// ---- POUs/Machine/CleaningStation/_VISU_CleanPU.TcVIS
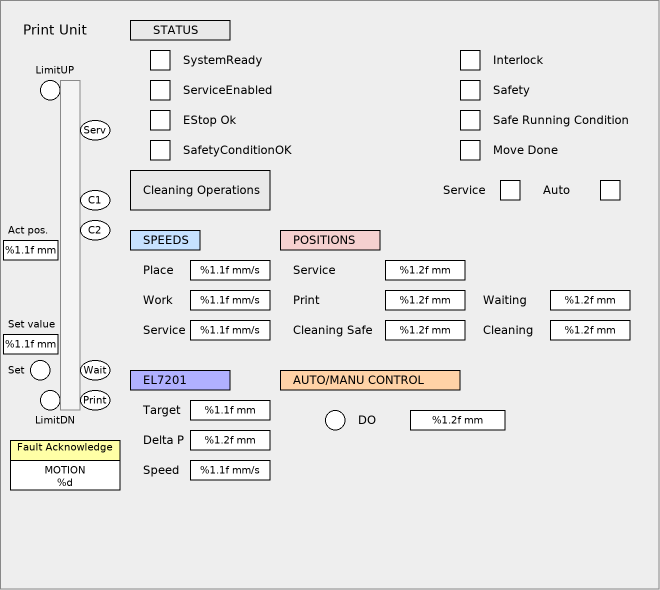
VISUALIZATION _VISU_CleanPU  // 660x590
VAR_IN_OUT
  mInst  : FB_CleaningMotorAxisPU;
END_VAR
    Rectangle (0,0 660x590)
    Polyline (200,380)
    Polyline (130,240)
    Rectangle (130,170 140x40)
    Rectangle (130,370 100x20)
    Rectangle (280,370 180x20)
    Rectangle (280,230 100x20)
    Rectangle (130,230 70x20)
    Rectangle (130,20 100x20)
    Rectangle (20,20 100x20), "Print Unit"
    Polyline (130,30)
    Polyline (230,30)
    Rectangle (150,20 60x20), "STATUS"
    RoundedRectangle (150,80 20x20), colour toggle: mInst.bI_UsrService
    RoundedRectangle (150,110 20x20), colour toggle: NOT mInst.bI_Emergency
    RoundedRectangle (150,140 20x20), colour toggle: mInst.bI_SafetyOk
    RoundedRectangle (460,140 20x20), colour toggle: NOT mInst.bL_Busy
    RoundedRectangle (150,50 20x20), colour toggle: mInst.bI_MachineReady
    Rectangle (180,50 120x20), "SystemReady"
    Rectangle (180,80 120x20), "ServiceEnabled"
    Rectangle (180,110 120x20), "EStop Ok"
    Rectangle (180,140 120x20), "SafetyConditionOK"
    Rectangle (490,140 90x20), "Move Done"
    Rectangle (290,370 170x20), "AUTO/MANU CONTROL"
    Polyline (450,380)
    Rectangle (30,60 50x20), "LimitUP"
    Ellipse (40,80 20x20), colour toggle: NOT mInst.bI_SensorTop
    Ellipse (40,390 20x20), colour toggle: NOT mInst.bI_SensorBottom
    Rectangle (30,410 50x20), "LimitDN"
    Scrollbar (60,80 20x330)
        p2245068023: 0.5
        p1057716461: mInst.fB_Axis.fO_ActualPosition
    Rectangle (140,230 70x20), "SPEEDS"
    Rectangle (190,260 80x20), "%1.1f mm/s", text variable: mInst.sI_SpeedDef.fP_PlaceSpeed
        OnMouseDown: write the text variable via VisuDialogs.Numpad
    Rectangle (190,290 80x20), "%1.1f mm/s", text variable: mInst.sI_SpeedDef.fP_WorkSpeed
        OnMouseDown: write the text variable via VisuDialogs.Numpad
    Rectangle (190,320 80x20), "%1.1f mm/s", text variable: mInst.sI_SpeedDef.fP_ServiceSpeed
        OnMouseDown: write the text variable via VisuDialogs.Numpad
    Rectangle (140,260 45x20), "Place"
    Rectangle (140,290 45x20), "Work"
    Rectangle (140,320 45x20), "Service"
        OnMouseDown: write the text variable via Edit
    Rectangle (290,260 90x20), "Service"
    Rectangle (290,290 90x20), "Print"
    Polyline (350,240)
    Rectangle (290,230 90x20), "POSITIONS"
    Rectangle (190,400 80x20), "%1.1f mm", text variable: 1000 * mInst.fB_Axis.fI_TargetPosition
    RoundedRectangle (460,80 20x20), colour toggle: mInst.bI_SafeToMove
    Rectangle (490,80 120x20), "Safety"
    RoundedRectangle (460,50 20x20), colour toggle: mInst.bI_SafeToMove
    Rectangle (490,50 120x20), "Interlock"
    Rectangle (5,360 25x20), "Set"
    Ellipse (30,360 20x20), colour toggle: mInst.fB_Axis.bI_SetPosition
        toggle mInst.fB_Axis.bI_SetPosition
    Rectangle (3,240 55x20), "%1.1f mm", text variable: 1000 * mInst.fB_Axis.fO_ActualPosition
    Rectangle (290,320 90x20), "Cleaning Safe"
    Rectangle (385,320 80x20), "%1.2f mm", text variable: mInst.fI_PositionClean1
        OnMouseDown: write the text variable via VisuDialogs.Numpad
    Rectangle (140,400 45x20), "Target"
    Rectangle (140,460 45x20), "Speed"
    Rectangle (190,460 80x20), "%1.1f mm/s", text variable: 1000 * mInst.fB_Axis.fI_SpeedLimit
    Rectangle (140,370 90x20), "EL7201"
    Rectangle (140,430 45x20), "Delta P"
    Rectangle (190,430 80x20), "%1.2f mm", text variable: 1000 * mInst.fB_Axis.fL_Delta_P
    Ellipse (80,120 30x20), "Serv", colour toggle: mInst.pInPosService
    Ellipse (80,220 30x20), "C2", colour toggle: mInst.pInPosClean2
    Ellipse (80,190 30x20), "C1", colour toggle: mInst.pInPosClean1
    Ellipse (80,360 30x20), "Wait", colour toggle: mInst.pInPosWait
    Ellipse (80,390 30x20), "Print", colour toggle: mInst.pInPosPrint
    Polyline (640,160)
    Rectangle (140,180 140x20), "Cleaning Operations"
    Polyline (270,200)
    RoundedRectangle (460,110 20x20), colour toggle: mInst.bL_SafeRunningCondition
    Rectangle (490,110 140x20), "Safe Running Condition"
    RoundedRectangle (600,180 20x20), colour toggle: mInst.bI_UsrAutoMode
    Rectangle (540,180 55x20), "Auto"
    Polyline (340,80)
    Rectangle (10,440 110x50), "Fault Acknowledge", colour toggle: (mInst.wL_ErrorCode) <> 0
    RoundedRectangle (10,460 110x30), "%d", text variable: mInst.wL_ErrorCode
        tap mInst.sADS_CleanAxis.bI_FaultAck
    RoundedRectangle (10,460 110x20), "MOTION"
    Rectangle (3,334 55x20), "%1.1f mm", text variable: mInst.fL_SetPositionValue
        OnMouseDown: write the text variable via VisuDialogs.Numpad
    Rectangle (480,320 65x20), "Cleaning"
    Rectangle (550,320 80x20), "%1.2f mm", text variable: mInst.fI_PositionClean2
        OnMouseDown: write the text variable via VisuDialogs.Numpad
    RoundedRectangle (500,180 20x20), colour toggle: mInst.bI_UsrService
    Rectangle (440,180 55x20), "Service"
    Rectangle (410,410 95x20), "%1.2f mm", text variable: mInst.sADS_CleanAxis.fI_ManualTargetPos
        OnMouseDown: write the text variable via VisuDialogs.Numpad, min mInst.sADS_CleanAxis.sO_AxisPosition.fC_Min, max mInst.sADS_CleanAxis.sO_AxisPosition.fC_Max
    Rectangle (355,410 50x20), "DO"
    Ellipse (325,410 20x20), colour toggle: mInst.sADS_CleanAxis.bI_ManualMove, input disabled if: NOT mInst.sADS_CleanAxis.bO_ManualMoveCanEx
        toggle mInst.sADS_CleanAxis.bI_ManualMove
    Rectangle (385,260 80x20), "%1.2f mm", text variable: mInst.fI_PositionService
        OnMouseDown: write the text variable via VisuDialogs.Numpad
    Rectangle (385,290 80x20), "%1.2f mm", text variable: mInst.fL_PrintPositionMM
        OnMouseDown: write the text variable via VisuDialogs.Numpad, min 0.8, max 2.5
    Rectangle (480,290 65x20), "Waiting"
    Rectangle (550,290 80x20), "%1.2f mm", text variable: mInst.fI_PositionWait
        OnMouseDown: write the text variable via VisuDialogs.Numpad
    Rectangle (5,314 50x20), "Set value"
    Rectangle (5,220 50x20), "Act pos."
END_VISUALIZATION

// ---- POUs/Machine/CleaningStation/_VISU_CleanSequence.TcVIS
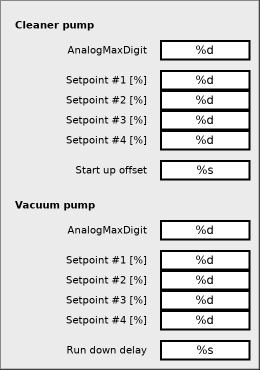
VISUALIZATION _VISU_CleanSequence  // 260x370
    Rectangle (0,0 260x370)
    Rectangle (160,40 90x20), "%d", text variable: PRG_MACHINE.fb_CleaningControl[PRG_MACHINE.iL_Sel_Module].fb_CleaningValvePump.lR_AnalogMaxDigitCleanerPump
        OnMouseDown: write the text variable via Default
    Rectangle (10,40 140x20), "AnalogMaxDigit"
    Rectangle (12,15 131x20), "Cleaner pump"
    Rectangle (160,70 90x20), "%d", text variable: PRG_MACHINE.fb_CleaningControl[PRG_MACHINE.iL_Sel_Module].fb_CleaningValvePump.lR_SetPoint1CleanerPump
        OnMouseDown: write the text variable via Default, min 0, max 100
    Rectangle (10,70 140x20), "Setpoint #1 [%]"
    Rectangle (160,90 90x20), "%d", text variable: PRG_MACHINE.fb_CleaningControl[PRG_MACHINE.iL_Sel_Module].fb_CleaningValvePump.lR_SetPoint2CleanerPump
        OnMouseDown: write the text variable via Default, min 0, max 100
    Rectangle (10,90 140x20), "Setpoint #2 [%]"
    Rectangle (160,110 90x20), "%d", text variable: PRG_MACHINE.fb_CleaningControl[PRG_MACHINE.iL_Sel_Module].fb_CleaningValvePump.lR_SetPoint3CleanerPump
        OnMouseDown: write the text variable via Default, min 0, max 100
    Rectangle (10,110 140x20), "Setpoint #3 [%]"
    Rectangle (160,130 90x20), "%d", text variable: PRG_MACHINE.fb_CleaningControl[PRG_MACHINE.iL_Sel_Module].fb_CleaningValvePump.lR_SetPoint4CleanerPump
        OnMouseDown: write the text variable via Default, min 0, max 100
    Rectangle (10,130 140x20), "Setpoint #4 [%]"
    Rectangle (160,220 90x20), "%d", text variable: PRG_MACHINE.fb_CleaningControl[PRG_MACHINE.iL_Sel_Module].fb_CleaningValvePump.lR_AnalogMaxDigitVacuumPump
        OnMouseDown: write the text variable via Default
    Rectangle (10,220 140x20), "AnalogMaxDigit"
    Rectangle (12,195 131x20), "Vacuum pump"
    Rectangle (160,250 90x20), "%d", text variable: PRG_MACHINE.fb_CleaningControl[PRG_MACHINE.iL_Sel_Module].fb_CleaningValvePump.lR_SetPoint1VacuumPump
        OnMouseDown: write the text variable via Default, min 0, max 100
    Rectangle (10,250 140x20), "Setpoint #1 [%]"
    Rectangle (160,270 90x20), "%d", text variable: PRG_MACHINE.fb_CleaningControl[PRG_MACHINE.iL_Sel_Module].fb_CleaningValvePump.lR_SetPoint2VacuumPump
        OnMouseDown: write the text variable via Default, min 0, max 100
    Rectangle (10,270 140x20), "Setpoint #2 [%]"
    Rectangle (160,290 90x20), "%d", text variable: PRG_MACHINE.fb_CleaningControl[PRG_MACHINE.iL_Sel_Module].fb_CleaningValvePump.lR_SetPoint3VacuumPump
        OnMouseDown: write the text variable via Default, min 0, max 100
    Rectangle (10,290 140x20), "Setpoint #3 [%]"
    Rectangle (160,310 90x20), "%d", text variable: PRG_MACHINE.fb_CleaningControl[PRG_MACHINE.iL_Sel_Module].fb_CleaningValvePump.lR_SetPoint4VacuumPump
        OnMouseDown: write the text variable via Default, min 0, max 100
    Rectangle (10,310 140x20), "Setpoint #4 [%]"
    Rectangle (160,160 90x20), "%s", text variable: PRG_MACHINE.fb_CleaningControl[PRG_MACHINE.iL_Sel_Module].fb_CleaningValvePump.tR_CleanerPumpOffset
        OnMouseDown: write the text variable via Default
    Rectangle (10,160 140x20), "Start up offset"
    Rectangle (160,340 90x20), "%s", text variable: PRG_MACHINE.fb_CleaningControl[PRG_MACHINE.iL_Sel_Module].fb_CleaningValvePump.tR_VacuumPumpDelay
        OnMouseDown: write the text variable via Default
    Rectangle (10,340 140x20), "Run down delay"
END_VISUALIZATION

// ---- POUs/Machine/EffectiveEncoderResolutionDetection/_VISU_EffectiveEncoderResolutionDetection.TcVIS
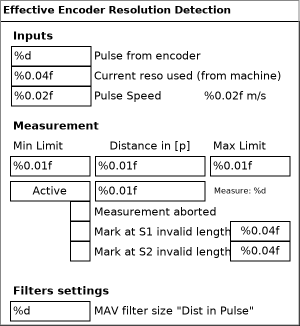
VISUALIZATION _VISU_EffectiveEncoderResolutionDetection  // 300x326
VAR_IN_OUT
	mInst : FB_EffectiveEncoderResolutionDetection;
END_VAR
    Rectangle (0,21 300x305)
    Rectangle (10,116 100x20), "Measurement"
    RoundedRectangle (10,181 80x20), "Active", colour toggle: mInst.bMeasurementActive
    Rectangle (95,156 110x20), "%0.01f", text variable: mInst.fDisInPulse
    Rectangle (95,136 110x20), "Distance in [p]"
    Rectangle (91,86 200x20), "Pulse Speed"
    Rectangle (11,86 80x20), "%0.02f", text variable: mInst.fSpeedPulse
    Rectangle (91,46 200x20), "Pulse from encoder"
    Rectangle (11,46 80x20), "%d", text variable: mInst.nPulse
    Rectangle (11,66 80x20), "%0.04f", text variable: mInst.fCurrentResolution, input disabled if: TRUE
    Rectangle (91,66 200x20), "Current reso used (from machine)"
    Rectangle (10,281 100x20), "Filters settings"
    Rectangle (91,301 200x20), "MAV filter size "Dist in Pulse""
    Rectangle (10,301 80x20), "%d", text variable: mInst.nDisInPulseFilterSz, input disabled if: TRUE
    Rectangle (10,26 100x20), "Inputs"
    Rectangle (0,0 240x20), "Effective Encoder Resolution Detection"
    Rectangle (211,181 80x20), "Measure: %d", tooltip "measurement counter", text variable: mInst.nMeasurementCounter
    Rectangle (10,156 80x20), "%0.01f", tooltip "Limits from machine", text variable: mInst.fEncoderPulseDistMin, colour toggle: mInst.bLower, input disabled if: TRUE
    Rectangle (210,156 80x20), "%0.01f", tooltip "Limits from machine", text variable: mInst.fEncoderPulseDistMax, colour toggle: mInst.bHigher, input disabled if: TRUE
    Rectangle (10,136 80x20), "Min Limit"
    Rectangle (210,136 80x20), "Max Limit"
    RoundedRectangle (70,201 20x20), colour toggle: mInst.bAborted
    Rectangle (91,202 200x20), "Measurement aborted"
    RoundedRectangle (70,221 20x20), colour toggle: mInst.bMarkInvalidLength_S1
    Rectangle (91,222 200x20), "Mark at S1 invalid length"
    RoundedRectangle (70,241 20x20), colour toggle: mInst.bMarkInvalidLength_S2
    Rectangle (91,242 200x20), "Mark at S2 invalid length"
    Rectangle (230,221 60x20), "%0.04f", tooltip "Mark length in [mm], minimum length=%0.02f [mm]", text variable: mInst.nMarkLength_S1/1000, colour toggle: mInst.bMarkInvalidLength_S1
        p4168582468: mInst.nC_MinMarkLength/1000
    Rectangle (230,241 60x20), "%0.04f", tooltip "Mark length in [mm], minimum length=%0.02f [mm]", text variable: mInst.nMarkLength_S2/1000, colour toggle: mInst.bMarkInvalidLength_S2
        p4168582468: mInst.nC_MinMarkLength/1000
    Rectangle (95,181 110x20), "%0.01f", text variable: mInst.nCurrentDistActive
    Rectangle (201,86 80x20), "%0.02f m/s", text variable: mInst.fSpeedUm_s/1_000_000, input disabled if: TRUE
END_VISUALIZATION

// ---- POUs/Machine/ExhaustSystem/_VISU_ExhaustSystemPrint.TcVIS
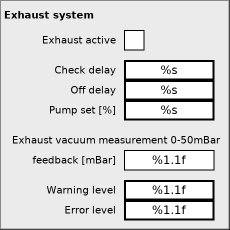
VISUALIZATION _VISU_ExhaustSystemPrint  // 230x230
VAR_IN_OUT
	mInst : FB_ExhaustSystemPrint;
END_VAR
    Rectangle (0,0 230x230)
    Rectangle (1,5 192x20), "Exhaust system"
    Rectangle (29,60 90x20), "Check delay"
    Rectangle (124,60 90x20), "%s", text variable: mInst.tR_VacuumCheckDelay
        OnMouseDown: write the text variable via Edit
    Rectangle (29,80 90x20), "Off delay"
    Rectangle (124,80 90x20), "%s", text variable: mInst.tR_FUOffDelay
        OnMouseDown: write the text variable via Edit
    RoundedRectangle (124,30 20x20), colour toggle: mInst.bO_FUActivate
    Rectangle (19,30 100x20), "Exhaust active"
    Rectangle (9,130 220x20), "Exhaust vacuum measurement 0-50mBar"
    Rectangle (29,150 90x20), "feedback [mBar]"
    Rectangle (124,150 90x20), "%1.1f", text variable: mInst.fL_VacuumAnalogLevelMBar
    Rectangle (29,180 90x20), "Warning level"
    Rectangle (124,180 90x20), "%1.1f", text variable: mInst.fR_VacuumWarningLevelMBar
        OnMouseDown: write the text variable via Edit
    Rectangle (29,200 90x20), "Error level"
    Rectangle (124,200 90x20), "%1.1f", text variable: mInst.fR_VacuumErrorLevelMBar
        OnMouseDown: write the text variable via Edit
    Rectangle (29,100 90x20), "Pump set [%]"
    Rectangle (124,100 90x20), "%s", text variable: mInst.iR_VacuumPumpSetPercent
        OnMouseDown: write the text variable via Edit, min 0, max 100
END_VISUALIZATION

// ---- POUs/Machine/PowerControl/_VISU_PowerControl.TcVIS
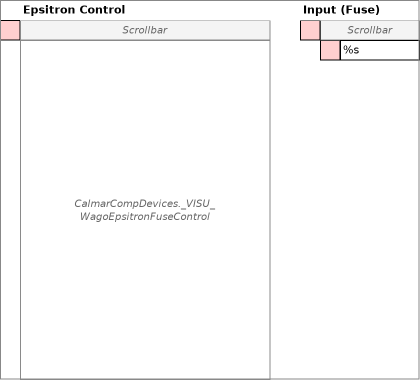
VISUALIZATION _VISU_PowerControl  // 420x380
VAR_IN_OUT
	mInst : FB_PowerControl;
END_VAR
    Frame (20,40 250x340)
        shows CalmarCompDevices._VISU_WagoEpsitronFuseControl(m_Inst_Fb := mInst.pEpsitronsInst[mInst.nEpsitronViewSel]^)
    RoundedRectangle (320,40 20x20), colour toggle: mInst.pFuseInputs[mInst.nFuseViewSel]^
    Scrollbar (320,20 100x20)
        p2245068023: mInst.nFuseInputsRegistered
        p1057716461: mInst.nFuseViewSel
    Rectangle (340,40 80x20), "%s", tooltip "%s", text variable: mInst.aFuseNames[mInst.nFuseViewSel]
        p4168582468: mInst.aFuseNames[mInst.nFuseViewSel]
    RoundedRectangle (300,20 20x20), tooltip "All Inputs ok", colour toggle: mInst.bO_AllFuseOk
    RoundedRectangle (0,20 20x20), tooltip "All Epsitron OK", colour toggle: mInst.bO_AllEpsitronOk
    Scrollbar (20,20 250x20)
        p2245068023: mInst.nEpsitronsRegistered
        p1057716461: mInst.nEpsitronViewSel
    Rectangle (20,0 250x20), "Epsitron Control"
    Rectangle (300,0 120x20), "Input (Fuse)"
END_VISUALIZATION

// ---- POUs/Machine/SheetDetectSupervision/VISU_SheetDetectSupervision.TcVIS
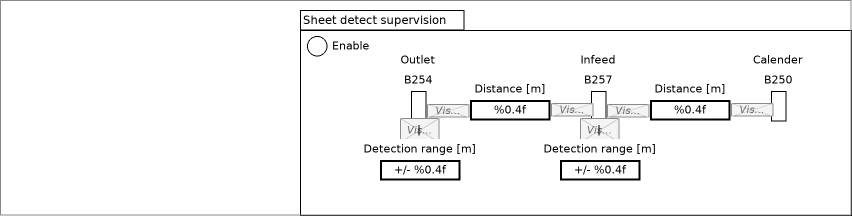
VISUALIZATION VISU_SheetDetectSupervision  // 852x216
VAR_IN_OUT
  mInst : FB_SheetDetectSupervision;
END_VAR
    Rectangle (300,10 164x20), "Sheet detect supervision"
    Rectangle (300,30 552x186)
    RoundedRectangle (771,91 15x30)
    Rectangle (756,70 45x20), "B250"
    RoundedRectangle (591,91 15x30)
    Rectangle (576,70 45x20), "B257"
    RoundedRectangle (411,91 15x30)
    Rectangle (396,70 45x20), "B254"
    Rectangle (650,100 80x20), "%0.4f", text variable: mInst.RemSheetDetectSupervisionPar.fR_SheetDetectDistance01
        OnMouseClick: write the text variable via Default
    Rectangle (650,79 80x20), "Distance [m]"
    Image (607,104 42x13), image: VisuSymbols.Symbols.ArrowBoldLeft
    Image (731,103 42x13), image: VisuSymbols.Symbols.ArrowBoldRight
    Rectangle (470,100 80x20), "%0.4f", text variable: mInst.RemSheetDetectSupervisionPar.fR_SheetDetectDistance02
        OnMouseClick: write the text variable via Default
    Rectangle (470,79 80x20), "Distance [m]"
    Image (427,104 42x13), image: VisuSymbols.Symbols.ArrowBoldLeft
    Image (551,103 42x13), image: VisuSymbols.Symbols.ArrowBoldRight
    Image (580,118 39x24), image: VisuSymbols.Symbols.DoubleArrow3
    Rectangle (560,160 80x20), "+/- %0.4f", text variable: mInst.RemSheetDetectSupervisionPar.fR_SheetDetectRange01_m
        OnMouseClick: write the text variable via Default
    Rectangle (540,139 120x20), "Detection range [m]"
    Line (599,135) (599,125)
    Rectangle (568,50 60x20), "Infeed"
    Rectangle (748,50 60x20), "Calender"
    Rectangle (388,50 60x20), "Outlet"
    Ellipse (307,36 20x20), tooltip "Reset"
        toggle mInst.RemSheetDetectSupervisionPar.bR_Enable
    Rectangle (329,36 60x20), "Enable"
    Image (400,118 39x24), image: VisuSymbols.Symbols.DoubleArrow3
    Rectangle (380,160 80x20), "+/- %0.4f", text variable: mInst.RemSheetDetectSupervisionPar.fR_SheetDetectRange02_m
        OnMouseClick: write the text variable via Default
    Rectangle (360,139 120x20), "Detection range [m]"
    Line (419,135) (419,125)
END_VISUALIZATION

// ---- POUs/Machine/UV_LED_Modul/_VISU_UvLedModule.TcVIS
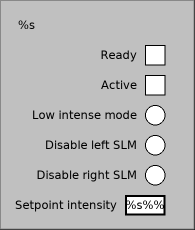
VISUALIZATION _VISU_UvLedModule  // 195x230
VAR_IN_OUT
  m_Inst_Fb   : FB_UvLedModule;
END_VAR
    Rectangle (0,0 195x230), colour variable: m_Inst_Fb._nColorRGB
        p2167032090: m_Inst_Fb._nColorRGB
        p3092690914: 16#FFFF0000
        p3450524324: 16#FF000000
    Rectangle (15,15 155x20), "%s", text variable: m_Inst_Fb._sColorName
    RoundedRectangle (145,45 20x20), colour toggle: m_Inst_Fb.IbReady
    Rectangle (20,45 120x20), "Ready"
    RoundedRectangle (145,75 20x20), colour toggle: m_Inst_Fb._bActivate
    Rectangle (20,75 120x20), "Active"
    Ellipse (145,105 20x20), colour toggle: m_Inst_Fb.RbLowIntenseMode
        toggle m_Inst_Fb.RbLowIntenseMode
    Rectangle (20,105 120x20), "Low intense mode"
    Ellipse (145,135 20x20), colour toggle: m_Inst_Fb.RbDisableLeft
        toggle m_Inst_Fb.RbDisableLeft
    Rectangle (20,135 120x20), "Disable left SLM"
    Ellipse (145,165 20x20), colour toggle: m_Inst_Fb.RbDisableRight
        toggle m_Inst_Fb.RbDisableRight
    Rectangle (20,165 120x20), "Disable right SLM"
    Rectangle (11,195 109x20), "Setpoint intensity"
    Rectangle (125,195 40x20), "%s%%", text variable: m_Inst_Fb.RnIntensitySetpoint
        OnMouseDown: write the text variable via VisuDialogs.Numpad, min m_Inst_Fb.CnMinIntensitySetpoint, max m_Inst_Fb.CnMaxIntensitySetpoint
END_VISUALIZATION

// ---- POUs/Print/Camera/LineCamera/_VISU_LineCamera.TcVIS
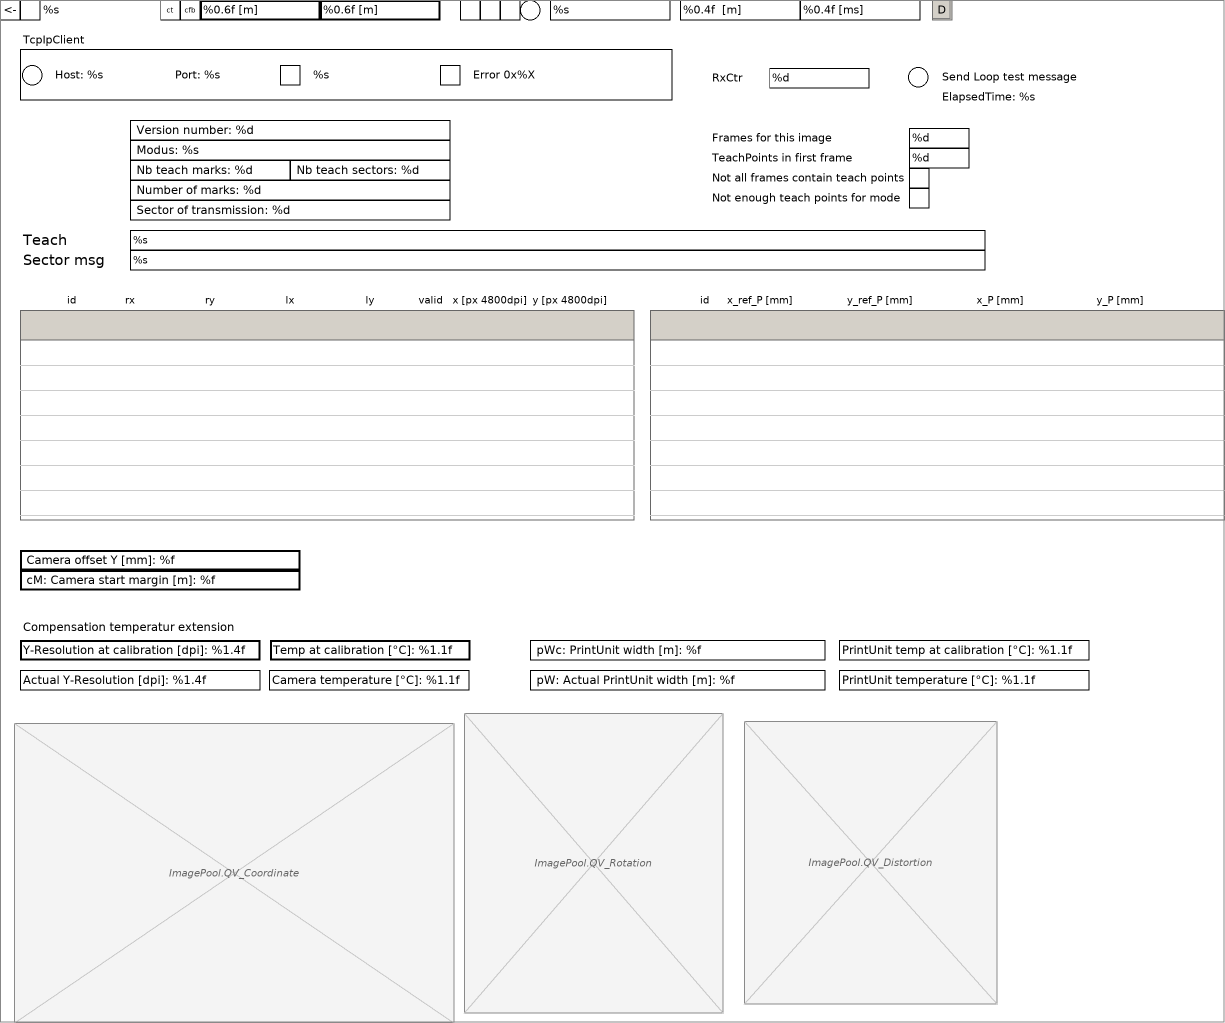
VISUALIZATION _VISU_LineCamera  // 1225x1023
VAR_INPUT
	m_Inst : FB_LineCamera;
END_VAR
    Rectangle (20,230 100x20), "Teach"
    Rectangle (130,230 855x20), "%s", text variable: m_Inst.sTeach
    Rectangle (130,120 320x20), "Version number: %d", text variable: m_Inst.nNbVersion
    Rectangle (130,160 160x20), "Nb teach marks: %d", text variable: m_Inst.nNbMarksTeach
    Table (20,310 614x210), data array: m_Inst.sCameraPoints
        p1128707560: GVL_Camera.cMaxNbMarks
        p2501879983: m_Inst.stCameraResult[INDEX].y_ref_Print
        p7306298: m_Inst.stCameraResult[INDEX].x_teach_Print
        p1933151965: m_Inst.stCameraResult[INDEX].y_teach_Print
        p3863566920: m_Inst.stCameraResult[INDEX].x_Print
        p2192122294: m_Inst.stCameraResult[INDEX].y_Print
        p3854506369: m_Inst.sCameraPoints[INDEX].id
        p1892666644: m_Inst.sCameraPoints[INDEX].x_ref
        p338671338: m_Inst.sCameraPoints[INDEX].y_ref
        p2170511999: m_Inst.sCameraPoints[INDEX].lx
        p3723444502: m_Inst.sCameraPoints[INDEX].ly
        p1218418051: m_Inst.sCameraPoints[INDEX].valid
    Rectangle (90,290 80x20), "rx"
    Rectangle (170,290 80x20), "ry"
    Rectangle (250,290 80x20), "lx"
    Rectangle (330,290 80x20), "ly"
    Rectangle (450,290 80x20), "x [px 4800dpi]"
    Rectangle (530,290 80x20), "y [px 4800dpi]"
    Rectangle (406,290 50x20), "valid"
    Rectangle (130,200 320x20), "Sector of transmission: %d", text variable: m_Inst.nSector
    Rectangle (530,640 295x20), "pWc: PrintUnit width [m]: %f", text variable: m_Inst._fPrintUnitWidthTC
    Image (14,723 440x300), image: ImagePool.QV_Coordinate
    Image (464,713 259x300), image: ImagePool.QV_Rotation
    Image (744,721 253x283), image: ImagePool.QV_Distortion
    Rectangle (20,250 100x20), "Sector msg"
    Rectangle (130,250 855x20), "%s", text variable: m_Inst.sMemLastMessage
    Rectangle (720,290 80x20), "x_ref_P [mm]"
    Rectangle (840,290 80x20), "y_ref_P [mm]"
    Rectangle (960,290 80x20), "x_P [mm]"
    Rectangle (1080,290 80x20), "y_P [mm]"
    Table (650,310 575x210), data array: m_Inst.sTeachPoints
        p1128707560: GVL_Camera.cMaxNbMarks
        p746581629: m_Inst.sTeachPoints[INDEX].y_Print
        p3104783080: m_Inst.stCameraResult[INDEX].x_ref_Print
        p2501879983: m_Inst.stCameraResult[INDEX].y_ref_Print
        p7306298: m_Inst.stCameraResult[INDEX].x_teach_Print
        p1933151965: m_Inst.stCameraResult[INDEX].y_teach_Print
        p3863566920: m_Inst.stCameraResult[INDEX].x_Print
        p2192122294: m_Inst.stCameraResult[INDEX].y_Print
        p3854506369: m_Inst.sTeachPoints[INDEX].id
        p1892666644: m_Inst.sTeachPoints[INDEX].x_ref_Print
        p338671338: m_Inst.sTeachPoints[INDEX].y_ref_Print
        p2170511999: m_Inst.sTeachPoints[INDEX].x_teach_Print
        p3723444502: m_Inst.sTeachPoints[INDEX].y_teach_Print
        p1218418051: m_Inst.sTeachPoints[INDEX].x_Print
    Rectangle (20,640 240x20), "Y-Resolution at calibration [dpi]: %1.4f", text variable: m_Inst.fCameraResolution
        OnMouseDown: write the text variable via Edit
    Rectangle (20,670 240x20), "Actual Y-Resolution [dpi]: %1.4f", text variable: m_Inst.fCameraRealResolution
    Rectangle (269,670 200x20), "Camera temperature [°C]: %1.1f", text variable: m_Inst.fCameraTemp
    Rectangle (270,640 200x20), "Temp at calibration [°C]: %1.1f", text variable: m_Inst.fCameraCalTemp
        OnMouseDown: write the text variable via Edit
    Rectangle (839,640 250x20), "PrintUnit temp at calibration [°C]: %1.1f", text variable: m_Inst._fPrintUnitCalTemp
    Rectangle (839,670 250x20), "PrintUnit temperature [°C]: %1.1f", text variable: m_Inst.fPrintUnitTemp
    Rectangle (20,617 245x20), "Compensation temperatur extension"
    Rectangle (530,670 295x20), "pW: Actual PrintUnit width [m]: %f", text variable: m_Inst.fPrintUnitWidthTAct
    Rectangle (130,180 320x20), "Number of marks: %d", text variable: m_Inst.nNbMarks
    Rectangle (20,550 280x20), "Camera offset Y [mm]: %f", text variable: m_Inst.fCameraAdjustmentY
        OnMouseDown: write the text variable via Edit
    Rectangle (20,570 280x20), "cM: Camera start margin [m]: %f", text variable: m_Inst.fCameraStartMargin
        OnMouseDown: write the text variable via Edit
    Rectangle (130,140 320x20), "Modus: %s", text variable: m_Inst.sModus
    Frame (0,0 861x79)
        shows _VISU_CameraTcpIp(m_Inst := m_Inst)
    Rectangle (290,160 160x20), "Nb teach sectors: %d", text variable: m_Inst.nNbSectorTeach
    Ellipse (908,67 20x20)
        tap m_Inst._bTestTx
    Rectangle (769,68 100x20), "%d", text variable: m_Inst.nRxMsg
    Rectangle (709,68 60x20), "RxCtr"
    Rectangle (939,67 161x20), "Send Loop test message"
    Rectangle (939,87 161x20), "ElapsedTime: %s", text variable: m_Inst._sTimeElapsed
    Rectangle (709,128 200x20), "Frames for this image"
    Rectangle (909,128 60x20), "%d", text variable: m_Inst.nNumFrames
    Rectangle (709,148 200x20), "TeachPoints in first frame"
    Rectangle (909,148 60x20), "%d", text variable: m_Inst.nNumPointsPerSectorT[1]
    Rectangle (709,168 200x20), "Not all frames contain teach points"
    RoundedRectangle (909,168 20x20), colour toggle: m_Inst.bNotAllFramesContainTeachPoints
    Rectangle (709,188 200x20), "Not enough teach points for mode"
    RoundedRectangle (909,188 20x20), colour toggle: m_Inst.bNotEnoughTeachPoints
    Rectangle (32,290 80x20), "id"
    Rectangle (690,290 30x20), "id"
END_VISUALIZATION

// ---- POUs/Print/Camera/MarkCameraWEU/_VISU_MarkCamera_WEU.TcVIS
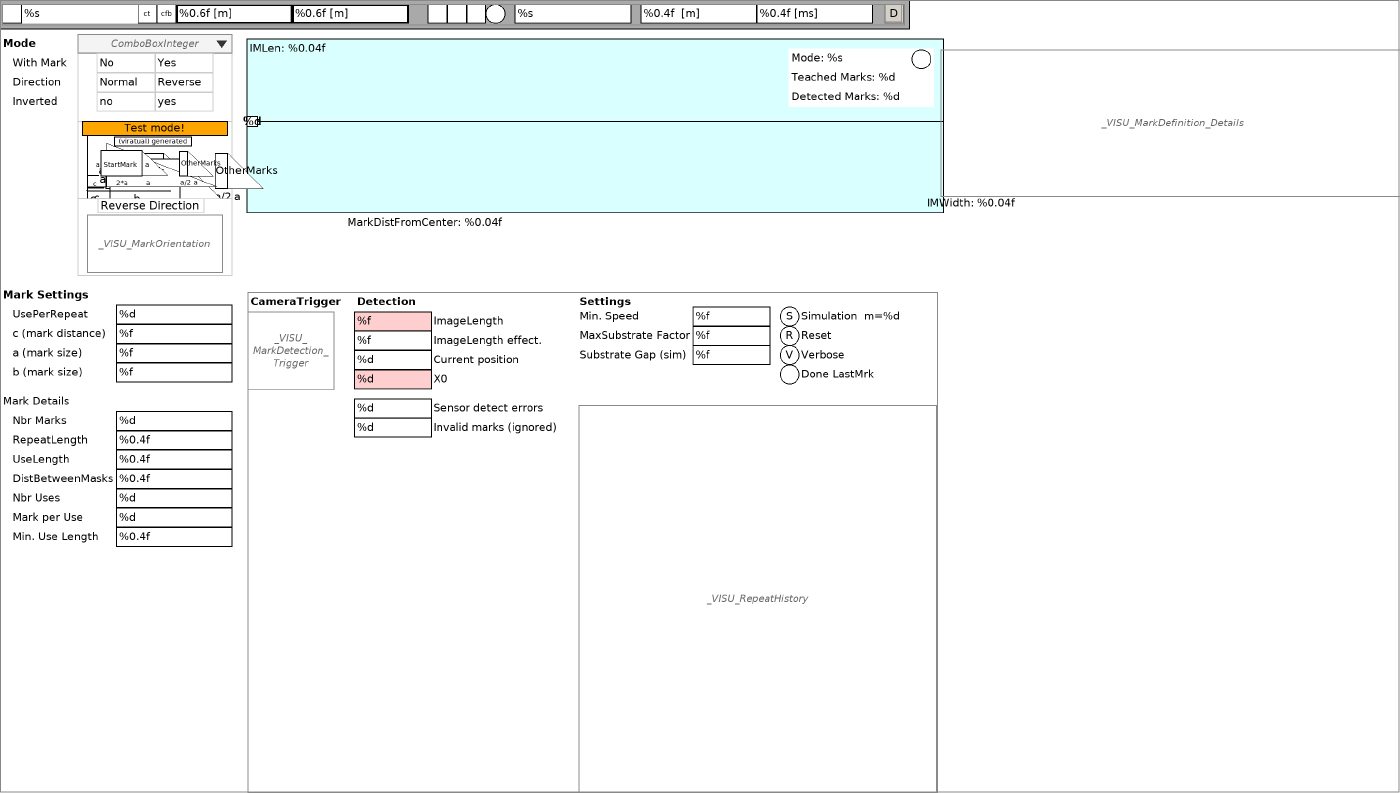
VISUALIZATION _VISU_MarkCamera_WEU  // 1447x820
VAR_IN_OUT
  mInst : FB_MarkCamera_WEU;
END_VAR
    RoundedRectangle (0,0 940x30)
    Frame (255,40 720x326)
        shows _VISU_MarkOverview(mInst := mInst)
    Frame (2,4 933x22)
        shows _VISU_CameraBase(m_Inst := mInst)
    Frame (0,35 241x543)
        shows _VISU_MarkModes(mInst := mInst)
    Frame (256,302 713x518)
        shows _VISU_MarkDetection(mInst := mInst.fbMarkDetection)
    Frame (942,51 505x143)
        shows _VISU_MarkDefinition(mInst := mInst.fbMarkDefinition)
END_VISUALIZATION

// ---- POUs/Print/Camera/MarkCameraWEU/_VISU_MarkDefinition.TcVIS
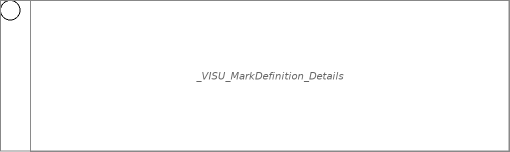
VISUALIZATION _VISU_MarkDefinition  // 510x152
VAR_IN_OUT
	mInst : FB_MarkDefinition;
END_VAR
    Ellipse (0,0 20x20), tooltip "Mark Details"
        toggle mInst.bShowDetail
    Frame (30,0 480x152), invisible if: NOT mInst.bShowDetail
        shows _VISU_MarkDefinition_Details(mInst := mInst)
END_VISUALIZATION

// ---- POUs/Print/Camera/MarkCameraWEU/_VISU_MarkDetection.TcVIS
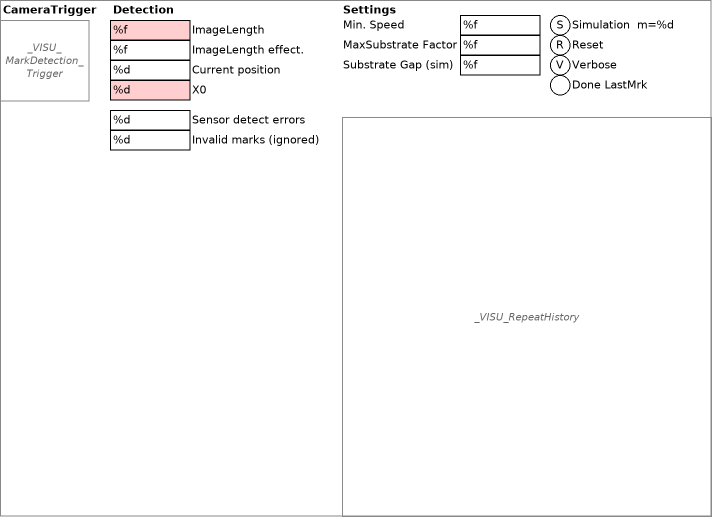
VISUALIZATION _VISU_MarkDetection  // 712x517
VAR_IN_OUT
	mInst: FB_MarkDetection;
END_VAR
    Ellipse (550,35 20x20), "R", tooltip "Reset"
        tap mInst.bManualReset
    Frame (0,20 89x81)
        shows _VISU_MarkDetection_Trigger(mInst := mInst)
    Rectangle (0,0 100x20), "CameraTrigger"
    Rectangle (110,20 80x20), "%f", text variable: mInst._fImageLength, colour toggle: mInst._fImageLength > 0
    Rectangle (189,20 140x20), "ImageLength"
    Rectangle (110,40 80x20), "%f", text variable: mInst._fImageLengthEffective
    Rectangle (189,40 140x20), "ImageLength effect."
    Rectangle (110,80 80x20), "%d", text variable: mInst._nX0, colour toggle: mInst._bValid
    Rectangle (189,80 140x20), "X0"
    Rectangle (110,60 80x20), "%d", text variable: mInst.nCurrentPos
    Rectangle (189,60 140x20), "Current position"
    Ellipse (550,15 20x20), "S", tooltip "Simulation"
        toggle mInst._bSimEnable
    Rectangle (569,15 100x20), "Simulation"
    Ellipse (550,75 20x20)
        toggle mInst.bR_TerminateLast
    Rectangle (569,75 100x20), "Done LastMrk"
    Rectangle (569,35 100x20), "Reset"
    Ellipse (550,55 20x20), "V", tooltip "Verbose"
        toggle mInst._bVerbose
    Rectangle (569,55 100x20), "Verbose"
    Rectangle (460,15 80x20), "%f", text variable: mInst.fC_MinimalSpeed, input disabled if: TRUE
    Rectangle (340,15 120x20), "Min. Speed"
    Rectangle (460,35 80x20), "%f", text variable: mInst.fC_MaxSubstrateFactor, input disabled if: TRUE
    Rectangle (340,35 120x20), "MaxSubstrate Factor"
    Rectangle (460,55 80x20), "%f", text variable: mInst._fSubstrateGap, invisible if: NOT mInst._bSimEnable
        OnMouseClick: write the text variable via Default
    Rectangle (340,55 120x20), "Substrate Gap (sim)", invisible if: NOT mInst._bSimEnable
    Rectangle (110,0 100x20), "Detection"
    Rectangle (340,0 100x20), "Settings"
    RoundedRectangle (110,110 80x20), "%d", text variable: mInst.nCtrSensorDetectError, colour toggle: mInst.nCtrSensorDetectError > 0
    Rectangle (189,110 140x20), "Sensor detect errors"
    RoundedRectangle (110,130 80x20), "%d", text variable: mInst.nCtrIgnoredMarks, colour toggle: mInst.nCtrIgnoredMarks > 0
    Rectangle (189,130 140x20), "Invalid marks (ignored)"
    TabControl (342,117 370x400)
        shows _VISU_RepeatHistory(mInst := mInst)
        shows _VISU_MarkHistory(mInst := mInst)
        [0]: TabTitle=Repeat History
        [1]: TabTitle=Mark History
    Rectangle (634,15 40x20), "m=%d", tooltip "simulation mode", text variable: mInst._nSimMode
        OnMouseClick: write the text variable via Default
END_VISUALIZATION

// ---- POUs/Print/Camera/MarkCameraWEU/_VISU_MarkHistory.TcVIS
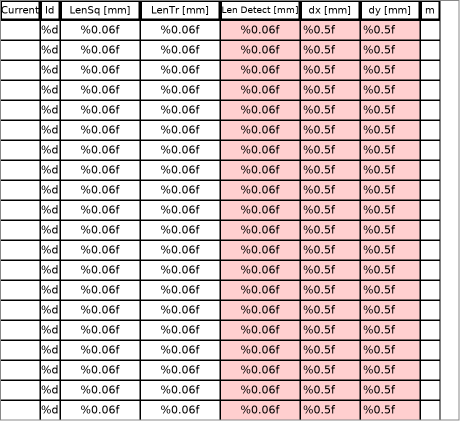
VISUALIZATION _VISU_MarkHistory  // 460x421
VAR_IN_OUT
	mInst : FB_MarkDetection;
END_VAR
    Frame (0,20 460x21)
        shows _VISU_MarkHistoryEntry(mInst := mInst.sMarkHistory[0])
    Rectangle (0,0 40x20), "Current"
    Rectangle (40,0 20x20), "Id"
    Rectangle (60,0 80x20), "LenSq [mm]"
    Rectangle (140,0 80x20), "LenTr [mm]"
    Rectangle (220,0 80x20), "Len Detect [mm]"
    Rectangle (300,0 60x20), "dx [mm]"
    Frame (0,40 460x21)
        shows _VISU_MarkHistoryEntry(mInst := mInst.sMarkHistory[1])
    Frame (0,60 460x21)
        shows _VISU_MarkHistoryEntry(mInst := mInst.sMarkHistory[2])
    Frame (0,80 460x21)
        shows _VISU_MarkHistoryEntry(mInst := mInst.sMarkHistory[3])
    Frame (0,100 460x21)
        shows _VISU_MarkHistoryEntry(mInst := mInst.sMarkHistory[4])
    Frame (0,120 460x21)
        shows _VISU_MarkHistoryEntry(mInst := mInst.sMarkHistory[5])
    Frame (0,140 460x21)
        shows _VISU_MarkHistoryEntry(mInst := mInst.sMarkHistory[6])
    Frame (0,160 460x21)
        shows _VISU_MarkHistoryEntry(mInst := mInst.sMarkHistory[7])
    Frame (0,180 460x21)
        shows _VISU_MarkHistoryEntry(mInst := mInst.sMarkHistory[8])
    Frame (0,200 460x21)
        shows _VISU_MarkHistoryEntry(mInst := mInst.sMarkHistory[9])
    Frame (0,220 460x21)
        shows _VISU_MarkHistoryEntry(mInst := mInst.sMarkHistory[10])
    Frame (0,240 460x21)
        shows _VISU_MarkHistoryEntry(mInst := mInst.sMarkHistory[11])
    Frame (0,260 460x21)
        shows _VISU_MarkHistoryEntry(mInst := mInst.sMarkHistory[12])
    Frame (0,280 460x21)
        shows _VISU_MarkHistoryEntry(mInst := mInst.sMarkHistory[13])
    Frame (0,300 460x21)
        shows _VISU_MarkHistoryEntry(mInst := mInst.sMarkHistory[14])
    Frame (0,320 460x21)
        shows _VISU_MarkHistoryEntry(mInst := mInst.sMarkHistory[15])
    Frame (0,340 460x21)
        shows _VISU_MarkHistoryEntry(mInst := mInst.sMarkHistory[16])
    Frame (0,360 460x21)
        shows _VISU_MarkHistoryEntry(mInst := mInst.sMarkHistory[17])
    Frame (0,380 460x21)
        shows _VISU_MarkHistoryEntry(mInst := mInst.sMarkHistory[18])
    Frame (0,400 460x21)
        shows _VISU_MarkHistoryEntry(mInst := mInst.sMarkHistory[19])
    Rectangle (360,0 60x20), "dy [mm]"
    Rectangle (420,0 20x20), "m", tooltip "missed"
END_VISUALIZATION

// ---- POUs/Print/Camera/MarkCameraWEU/_VISU_MarkHistoryEntry.TcVIS
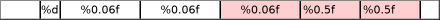
VISUALIZATION _VISU_MarkHistoryEntry  // 440x20
VAR_IN_OUT
	mInst : ST_MarkDefinition;
END_VAR
    Rectangle (220,0 200x20), colour toggle: mInst.sState.bSet
    RoundedRectangle (0,0 40x20), colour variable: mInst.sView.colorFill
    Rectangle (40,0 20x20), "%d", text variable: mInst.nId, colour toggle: mInst.nId=1
    Rectangle (60,0 80x20), "%0.06f", tooltip "square length [mm]", text variable: mInst.fSqLength * 1000
        p4168582468: mInst.fSqLength * 1000
    Rectangle (140,0 80x20), "%0.06f", tooltip "triangle length [mm]", text variable: mInst.fTrLength * 1000
        p4168582468: mInst.fTrLength
    Rectangle (220,0 80x20), "%0.06f", tooltip "detected length [mm]", text variable: mInst.sState.fLengthReal * 1000, colour toggle: mInst.sState.bSet
    Rectangle (300,0 60x20), "%0.5f", text variable: minst.sState.dx * 1000, colour toggle: mInst.sState.bSet
    Rectangle (360,0 60x20), "%0.5f", text variable: minst.sState.dy * 1000, colour toggle: mInst.sState.bSet
    RoundedRectangle (420,0 20x20), tooltip "missed mark", colour toggle: mInst.sState.bMissed, colour variable: mInst.sView.colorFill
END_VISUALIZATION

// ---- POUs/Print/Camera/MarkCameraWEU/_VISU_MarkModes.TcVIS
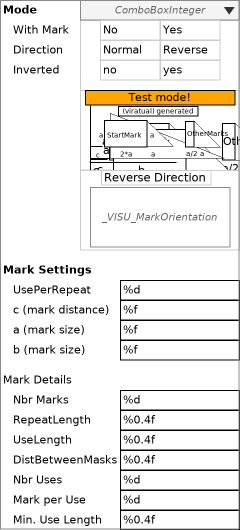
VISUALIZATION _VISU_MarkModes  // 240x530
VAR_IN_OUT
  mInst : FB_MarkCamera_WEU;
END_VAR
    Rectangle (80,20 160x80)
    Rectangle (80,90 160x80)
    Rectangle (0,0 120x20), "Mode"
    Rectangle (120,300 120x20), "%f", text variable: mInst.fMarkSpec_c
        OnMouseClick: write the text variable via Default
    Rectangle (120,280 120x20), "%d", text variable: mInst.nUsePerRepeat
        OnMouseClick: write the text variable via Default
    Rectangle (10,280 110x20), "UsePerRepeat"
    Rectangle (10,320 110x20), "a (mark size)", input disabled if: TRUE
    Rectangle (10,300 110x20), "c (mark distance)", input disabled if: TRUE
    Rectangle (120,320 120x20), "%f", text variable: mInst.fMarkSpec_a, colour toggle: mInst.fMarkSpec_a = 0
        OnMouseClick: write the text variable via Default
    ComboBoxInteger (80,0 160x20), variable: mInst.eMarkMode, text list: 'TL_MarkMode'
    Rectangle (10,340 110x20), "b (mark size)", input disabled if: TRUE
    Rectangle (120,340 120x20), "%f", text variable: mInst.fMarkSpec_b
        OnMouseClick: write the text variable via Default
    Group (90,95 147x63), invisible if: mInst.eMarkMode <> E_MarkMode.AutoDefault
        Polyline (0,0) (0,84) (121,84)
        Polygon (79,28) (79,65) (117,65)
        Rectangle (19,28 60x37)
        Rectangle (37,64 26x19), "2*a"
        Rectangle (81,64 37x19), "a"
        Rectangle (9,37 26x19), "a"
        Rectangle (19,37 61x19), "StartMark"
        Line (1,64) (17,64)
        Rectangle (4,65 26x19), "c"
        Rectangle (79,37 26x19), "a"
        Group (129,28 76x55)
            Rectangle (3,0 13x37)
            Polygon (16,0) (16,37) (53,37)
            Rectangle (0,36 26x19), "a/2"
            Rectangle (1,9 75x19), "OtherMarks"
            Rectangle (20,36 37x19), "a"
    Group (90,95 113x65), invisible if: mInst.eMarkMode <> E_MarkMode.OneDefault
        Polyline (0,0) (0,103) (147,103)
        Polygon (95,33) (95,78) (141,78)
        Rectangle (23,34 73x45)
        Rectangle (45,78 32x23), "2*a"
        Rectangle (97,78 45x23), "a"
        Rectangle (10,44 32x23), "a"
        Rectangle (23,44 75x23), "StartMark"
        Line (1,78) (21,78)
        Rectangle (0,78 32x23), "c"
        Rectangle (96,44 32x23), "a"
    Group (90,95 100x60), invisible if: mInst.eMarkMode <> E_MarkMode.OneTriangle
        Polyline (0,0) (0,89) (146,89)
        Polygon (20,18) (20,63) (134,63)
        Rectangle (45,64 33x23), "b"
        Rectangle (11,36 33x23), "a"
        Rectangle (23,36 76x23), "StartMark"
        Line (0,63) (19,63)
        Rectangle (0,64 33x23), "c"
    RoundedRectangle (100,40 60x20), "Normal", colour toggle: NOT mInst.bPrintDirReverse
    Rectangle (10,40 110x20), "Direction"
    RoundedRectangle (160,40 60x20), "Reverse", colour toggle: mInst.bPrintDirReverse
    Rectangle (10,20 110x20), "With Mark"
    RoundedRectangle (100,20 60x20), "No", colour toggle: NOT mInst.bPrintMarkExist
    RoundedRectangle (160,20 60x20), "Yes", colour toggle: mInst.bPrintMarkExist
    Rectangle (10,60 110x20), "Inverted", tooltip "Mark is flipped/inverted"
    RoundedRectangle (160,60 60x20), "yes", colour toggle: mInst.bMarkInverted
    RoundedRectangle (100,60 60x20), "no", colour toggle: NOT mInst.bMarkInverted
    Rectangle (80,170 160x80)
    RoundedRectangle (85,90 150x15), "Test mode!", invisible if: mInst.eMarkMode = E_MarkMode.AutoDefault OR mInst.eMarkMode = E_MarkMode.None
    Rectangle (0,260 120x20), "Mark Settings"
    Frame (90,187 140x60)
        shows _VISU_MarkOrientation(mInst := mInst)
    RoundedRectangle (101,170 110x15), "Reverse Direction"
        toggle mInst.bPrintDirReverse
    Rectangle (10,410 110x20), "RepeatLength"
    Rectangle (120,410 120x20), "%0.4f", text variable: mInst.fbMarkDefinition._fImageLength, colour toggle: mInst._bImageLengthError, input disabled if: TRUE
    Rectangle (0,370 120x20), "Mark Details"
    Rectangle (10,430 110x20), "UseLength"
    Rectangle (120,430 120x20), "%0.4f", text variable: mInst.fbMarkDefinition._fUseLength, input disabled if: TRUE
    Rectangle (10,450 110x20), "DistBetweenMasks"
    Rectangle (120,450 120x20), "%0.4f", text variable: mInst.fbMarkDefinition._fDistBetweenMarks, input disabled if: TRUE
    Rectangle (10,470 110x20), "Nbr Uses"
    Rectangle (120,470 120x20), "%d", text variable: mInst.fbMarkDefinition._nUses, input disabled if: TRUE
    Rectangle (10,490 110x20), "Mark per Use"
    Rectangle (120,490 120x20), "%d", text variable: mInst.fbMarkDefinition._nMarksPerUse, input disabled if: TRUE
    Rectangle (10,390 110x20), "Nbr Marks"
    Rectangle (120,390 120x20), "%d", tooltip "teached marks", text variable: mInst.fbMarkDefinition._nMarks, colour toggle: mInst.fbMarkDefinition._nMarks = 0, input disabled if: TRUE
    Rectangle (10,510 110x20), "Min. Use Length"
    Rectangle (120,510 120x20), "%0.4f", text variable: mInst.fbMarkDefinition.fC_MinUseLength, input disabled if: TRUE
    Group (90,106 147x56), invisible if: mInst.eMarkMode <> E_MarkMode.None
        Polyline (0,1) (0,56) (86,56)
        Polygon (56,14) (56,40) (83,40)
        Rectangle (14,14 43x27)
        Rectangle (27,41 19x14), "2*a"
        Rectangle (58,41 27x14), "a"
        Rectangle (6,22 19x14), "a"
        Rectangle (14,22 44x14), "StartMark"
        Line (0,40) (12,40)
        Rectangle (3,42 19x14), "c"
        Rectangle (57,22 19x14), "a"
        Rectangle (95,15 9x26)
        Polygon (104,15) (104,41) (130,41)
        Rectangle (93,41 18x13), "a/2"
        Rectangle (94,21 53x13), "OtherMarks"
        Rectangle (107,41 26x13), "a"
        Rectangle (28,0 80x10), "(viratual) generated"
END_VISUALIZATION

// ---- POUs/Print/Camera/MarkCameraWEU/_VISU_MarkOverview.TcVIS
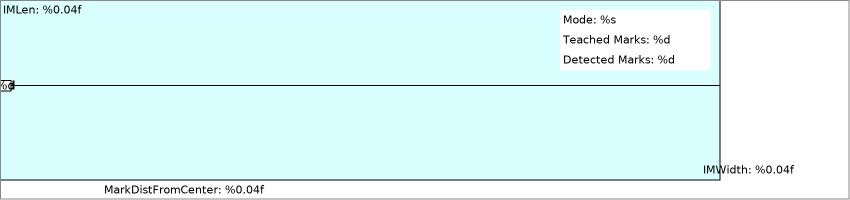
VISUALIZATION _VISU_MarkOverview  // 850x200
VAR_IN_OUT
  mInst : FB_MarkCamera_WEU;
END_VAR
    Rectangle (0,0 720x180)
    Rectangle (0,0 150x20), "IMLen: %0.04f", text variable: mInst._fImageLength
    Rectangle (700,160 150x20), "IMWidth: %0.04f", text variable: mInst._fImageWidth
        p2858320360: -90
    Line (0,85) (720,85)
    Rectangle (101,180 220x20), "MarkDistFromCenter: %0.04f", text variable: mInst.fMarkDistFromCenter
        p2858320360: -90
    Frame (0,80 11x11)
        shows _VISU_MarkViewMini(mInst := mInst.fbMarkDefinition.sMarkDef[1])
    Frame (0,80 11x11)
        shows _VISU_MarkViewMini(mInst := mInst.fbMarkDefinition.sMarkDef[2])
    Frame (0,80 11x11)
        shows _VISU_MarkViewMini(mInst := mInst.fbMarkDefinition.sMarkDef[3])
    Frame (0,80 11x11)
        shows _VISU_MarkViewMini(mInst := mInst.fbMarkDefinition.sMarkDef[4])
    Frame (0,80 11x11)
        shows _VISU_MarkViewMini(mInst := mInst.fbMarkDefinition.sMarkDef[5])
    Frame (0,80 11x11)
        shows _VISU_MarkViewMini(mInst := mInst.fbMarkDefinition.sMarkDef[6])
    Frame (0,80 11x11)
        shows _VISU_MarkViewMini(mInst := mInst.fbMarkDefinition.sMarkDef[7])
    Frame (0,80 11x11)
        shows _VISU_MarkViewMini(mInst := mInst.fbMarkDefinition.sMarkDef[8])
    Frame (0,80 11x11)
        shows _VISU_MarkViewMini(mInst := mInst.fbMarkDefinition.sMarkDef[9])
    Frame (0,80 11x11)
        shows _VISU_MarkViewMini(mInst := mInst.fbMarkDefinition.sMarkDef[10])
    Frame (0,80 11x11)
        shows _VISU_MarkViewMini(mInst := mInst.fbMarkDefinition.sMarkDef[11])
    Frame (0,80 11x11)
        shows _VISU_MarkViewMini(mInst := mInst.fbMarkDefinition.sMarkDef[12])
    Frame (0,80 11x11)
        shows _VISU_MarkViewMini(mInst := mInst.fbMarkDefinition.sMarkDef[13])
    Frame (0,80 11x11)
        shows _VISU_MarkViewMini(mInst := mInst.fbMarkDefinition.sMarkDef[15])
    Frame (0,80 11x11)
        shows _VISU_MarkViewMini(mInst := mInst.fbMarkDefinition.sMarkDef[18])
    Frame (0,80 11x11)
        shows _VISU_MarkViewMini(mInst := mInst.fbMarkDefinition.sMarkDef[16])
    Frame (0,80 11x11)
        shows _VISU_MarkViewMini(mInst := mInst.fbMarkDefinition.sMarkDef[17])
    Frame (0,80 11x11)
        shows _VISU_MarkViewMini(mInst := mInst.fbMarkDefinition.sMarkDef[19])
    Frame (0,80 11x11)
        shows _VISU_MarkViewMini(mInst := mInst.fbMarkDefinition.sMarkDef[20])
    Frame (0,80 11x11)
        shows _VISU_MarkViewMini(mInst := mInst.fbMarkDefinition.sMarkDef[21])
    Frame (0,80 11x11)
        shows _VISU_MarkViewMini(mInst := mInst.fbMarkDefinition.sMarkDef[22])
    Frame (0,80 11x11)
        shows _VISU_MarkViewMini(mInst := mInst.fbMarkDefinition.sMarkDef[23])
    Frame (0,80 11x11)
        shows _VISU_MarkViewMini(mInst := mInst.fbMarkDefinition.sMarkDef[24])
    Frame (0,80 11x11)
        shows _VISU_MarkViewMini(mInst := mInst.fbMarkDefinition.sMarkDef[25])
    Frame (0,80 11x11)
        shows _VISU_MarkViewMini(mInst := mInst.fbMarkDefinition.sMarkDef[26])
    Frame (0,80 11x11)
        shows _VISU_MarkViewMini(mInst := mInst.fbMarkDefinition.sMarkDef[27])
    Frame (0,80 11x11)
        shows _VISU_MarkViewMini(mInst := mInst.fbMarkDefinition.sMarkDef[28])
    Frame (0,80 11x11)
        shows _VISU_MarkViewMini(mInst := mInst.fbMarkDefinition.sMarkDef[29])
    Frame (0,80 11x11)
        shows _VISU_MarkViewMini(mInst := mInst.fbMarkDefinition.sMarkDef[30])
    Rectangle (560,30 150x20), "Teached Marks: %d", text variable: mInst._nTeachedPoints, colour toggle: mInst._bTeachOk
    Rectangle (560,50 150x20), "Detected Marks: %d", text variable: mInst._nDetectedMarks, colour toggle: mInst._nDetectedMarks = mInst._nTeachedPoints AND mInst._nTeachedPoints > 0
    Rectangle (560,10 150x20), "Mode: %s", text variable: mInst.eMarkMode
    Frame (0,80 11x11)
        shows _VISU_MarkViewMini(mInst := mInst.fbMarkDefinition.sMarkDef[14])
END_VISUALIZATION

// ---- POUs/Print/Camera/MarkCameraWEU/_VISU_MarkViewMini.TcVIS
VISUALIZATION _VISU_MarkViewMini  // 10x10
VAR_IN_OUT
	mInst : ST_MarkDefinition;
END_VAR
    RoundedRectangle (0,0 10x10), "%d", text variable: mInst.nId, invisible if: NOT mInst.sView.bShow, colour variable: mInst.sView.colorFill
        p3560616238: mInst.sView.nXPosPx
        p2738717112: mInst.sView.nYPosPx
END_VISUALIZATION

// ---- POUs/Print/Camera/MarkCameraWEU/_VISU_RepeatHistoryEntry.TcVIS
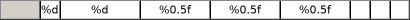
VISUALIZATION _VISU_RepeatHistoryEntry  // 410x20
VAR_IN_OUT
	mInst : ST_RepeatHistory;
END_VAR
    RoundedRectangle (0,0 40x20), colour toggle: mInst.bSelected
    Rectangle (40,0 20x20), "%d", text variable: mInst.nIndex
    Rectangle (60,0 80x20), "%d", tooltip "X0 [SubPx]", text variable: mInst.nX0
    Rectangle (140,0 70x20), "%0.5f", tooltip "Length Effective", text variable: mInst.fLenEffective
    Rectangle (210,0 70x20), "%0.5f", tooltip "Length Configured", text variable: mInst.fLen
    Rectangle (280,0 70x20), "%0.5f", tooltip "Length diff", text variable: mInst.fLenDiff
    RoundedRectangle (350,0 20x20), tooltip "Length not in range", colour toggle: mInst.bLenNotInRange
    RoundedRectangle (370,0 20x20), tooltip "invalid & ignored marks", colour toggle: mInst.bInvalidIngoredMarks
    RoundedRectangle (390,0 20x20), tooltip "missing marks", colour toggle: mInst.bMissingMarks
END_VISUALIZATION

// ---- POUs/Print/Camera/_VISU_CameraBase.TcVIS
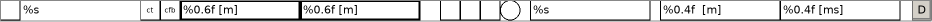
VISUALIZATION _VISU_CameraBase  // 932x22
VAR_IN_OUT
	m_Inst : FB_CameraBase;
END_VAR
    Rectangle (660,0 120x20), "%0.4f [m]", tooltip "TriggerDistance", text variable: m_Inst._fTriggerDistance
        OnMouseDown: write the text variable via Default
    Rectangle (780,0 120x20), "%0.4f [ms]", tooltip "TriggerPulseLength", text variable: m_Inst._fTriggerPulseLength
        OnMouseDown: write the text variable via Default
    RoundedRectangle (440,0 20x20), tooltip "Initialized", colour toggle: m_Inst._bInitialized
    RoundedRectangle (460,0 20x20), tooltip "Camera sink", colour toggle: m_Inst._iCameraSink <> 0
    RoundedRectangle (480,0 20x20), tooltip "Camera trigger", colour toggle: m_Inst._iCameraTrigger <> 0
    Ellipse (500,0 20x20), tooltip "simulate"
        toggle m_Inst._bSimulate
    Frame (0,0 432x22)
        shows _VISU_CameraBaseSetting(m_Inst := m_Inst)
    Button (912,0 20x20), "D", tooltip "Camera Detail: %s", invisible if: m_Inst._sVisuName='unvailable'
        p4168582468: m_Inst._sVisuName
        OnMouseClick: change screen: AssignExpression m_Inst._sVisuName
    Rectangle (530,0 120x20), "%s", tooltip "configured camera mode, active=%s", text variable: m_Inst._eCameraMode
        p4168582468: m_Inst.eCameraMode
        OnMouseDown: write the text variable via Default
END_VISUALIZATION

// ---- POUs/Print/Camera/_VISU_CameraBaseSetting.TcVIS
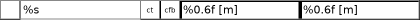
VISUALIZATION _VISU_CameraBaseSetting  // 420x20
VAR_IN_OUT
	m_Inst : FB_CameraBase;
END_VAR
    Rectangle (300,0 120x20), "%0.6f [m]", tooltip "CameraToPrintUnit", text variable: m_Inst._fCameraToPrintOffset
        OnMouseDown: write the text variable via Default
    Rectangle (180,0 120x20), "%0.6f [m]", tooltip "DetectToCamera", text variable: m_Inst._fDetectToCameraOffset
        OnMouseDown: write the text variable via Default
    RoundedRectangle (140,0 20x20), "ct", tooltip "UseCameraTrigger", colour toggle: m_Inst._bUseCameraTrigger
    RoundedRectangle (160,0 20x20), "cfb", tooltip "UseCameraTriggerFeedback", colour toggle: m_Inst._bUseCameraTriggerFeedback
    Rectangle (20,0 120x20), "%s", text variable: m_Inst.sName, colour toggle: m_Inst._bActivated <> 0
    RoundedRectangle (0,0 20x20), tooltip "Camera activated", colour toggle: m_Inst._bActivated <> 0
END_VISUALIZATION

// ---- POUs/Print/Camera/_VISU_CameraTcpIp.TcVIS
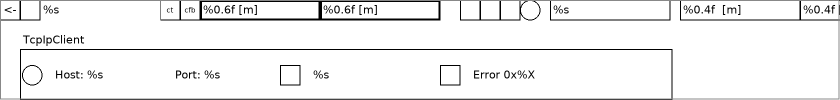
VISUALIZATION _VISU_CameraTcpIp  // 840x100
VAR_IN_OUT
	m_Inst : FB_CameraTcpIp;
END_VAR
    Rectangle (20,49 652x51)
    Frame (20,0 820x23)
        shows _VISU_CameraBase(m_Inst := m_Inst)
    Frame (22,65 240x21)
        shows _VISU_CameraTcpIpSetting(m_Inst := m_Inst)
    RoundedRectangle (0,0 20x20), "<-"
        OnMouseClick: change screen: Previous 
    RoundedRectangle (280,65 20x20), tooltip "Connected", colour toggle: m_Inst._pFbTcpIpClient^.bConnected
    RoundedRectangle (440,65 20x20), tooltip "Error", colour toggle: m_Inst._bConnectionError
    Rectangle (310,65 120x20), "%s", text variable: m_Inst._pFbTcpIpClient^.eStep
    Rectangle (470,65 120x20), "Error 0x%X", text variable: m_Inst._pFbTcpIpClient^.nErrId
    Rectangle (20,30 120x20), "TcpIpClient"
END_VISUALIZATION

// ---- POUs/Print/Camera/_VISU_CameraTcpIpSetting.TcVIS
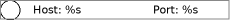
VISUALIZATION _VISU_CameraTcpIpSetting  // 230x20
VAR_IN_OUT
	m_Inst : FB_CameraTcpIp;
END_VAR
    Ellipse (0,0 20x20)
        toggle m_Inst._pFbTcpIpClient^.bEnable
    Rectangle (30,0 120x20), "Host: %s", tooltip "Camera ip address", text variable: m_Inst._pFbTcpIpClient^.sRemoteHost
    Rectangle (150,0 80x20), "Port: %s", tooltip "camera port", text variable: m_Inst._pFbTcpIpClient^.nRemotePort
END_VISUALIZATION

// ---- POUs/Print/Camera/_VISU_CameraTrigger.TcVIS
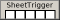
VISUALIZATION _VISU_CameraTrigger  // 60x20
VAR_IN_OUT
	mInst : FB_CameraTrigger;
END_VAR
    RoundedRectangle (0,0 60x20), tooltip "Trigger Armed", colour toggle: mInst.bTriggerArmed
    RoundedRectangle (15,10 10x10), tooltip "Speed valid", colour toggle: mInst.bSpeedValid
    RoundedRectangle (25,10 10x10), tooltip "AutomaticMode or ManualTeach", colour toggle: mInst._bCamManualTeachMode OR mInst.bI_AutomaticMode
    RoundedRectangle (35,10 10x10), tooltip "Inhibit trigger", colour toggle: NOT mInst.bInhibitTrigger
    RoundedRectangle (45,10 10x10), tooltip "HwEnable", colour toggle: mInst.bI_HwEnable
    RoundedRectangle (5,10 10x10), tooltip "Init ok", colour toggle: mInst.bInitOk
    Rectangle (0,0 60x10), "SheetTrigger", tooltip "SheetDetect"
END_VISUALIZATION

// ---- POUs/Print/Camera/_VISU_DeformationPoint.TcVIS
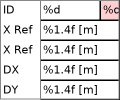
VISUALIZATION _VISU_DeformationPoint  // 120x100
VAR_IN_OUT
	m_Inst : ST_DeformationPointAccurate;
END_VAR
    Rectangle (40,0 60x20), "%d", text variable: m_Inst.index
    Rectangle (0,0 40x20), "ID"
    Rectangle (40,20 80x20), "%1.4f [m]", text variable: m_Inst.x_ref
    Rectangle (0,20 40x20), "X Ref"
    Rectangle (40,40 80x20), "%1.4f [m]", text variable: m_Inst.y_ref
    Rectangle (0,40 40x20), "X Ref"
    Rectangle (40,60 80x20), "%1.4f [m]", text variable: m_Inst.dx
    Rectangle (0,60 40x20), "DX"
    Rectangle (40,80 80x20), "%1.4f [m]", text variable: m_Inst.dy
    Rectangle (0,80 40x20), "DY"
    Rectangle (100,0 20x20), "%d", text variable: m_Inst.valid
END_VISUALIZATION

// ---- POUs/Print/Camera/_VISU_SystronCamera.TcVIS
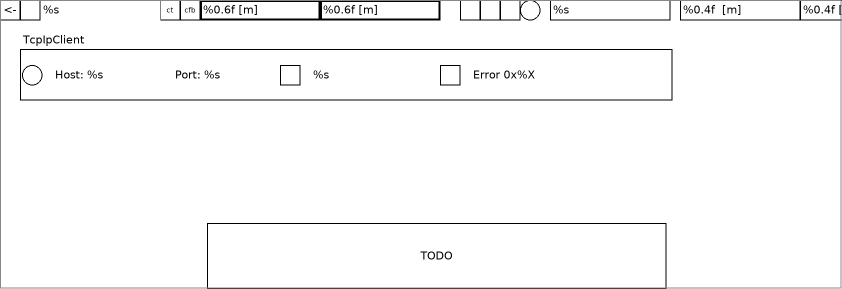
VISUALIZATION _VISU_SystronCamera  // 842x289
    Rectangle (207,223 459x66), "TODO"
    Frame (0,0 842x135)
        shows _VISU_CameraTcpIp(m_Inst := PRG_PRINT.fbLineCamera)
END_VISUALIZATION

// ---- POUs/Print/DefGrid/_Test/Txt_GridTypeSelection.TcTLO
TEXTLIST Txt_GridTypeSelection
  0 = 'Default (dy from StartMark)'
  1 = 'None: Grid calculated dx/dy=0'
  2 = 'Test_AllDxFactor'
  3 = 'Test_AllDyFactor'
  4 = 'Test_DxColFactor'
  5 = 'Test_DyColFactro'
  6 = 'Test_Dx_FirstRowOnlyFactor'
   = ''
END_TEXTLIST

// ---- POUs/Print/DefGrid/_VISU_Templates/E_DeformationType.TcTLO
TEXTLIST E_DeformationType
  0 = 'NoDeformation'
  1 = 'ScriptGrid'
  2 = 'ScriptGridTrend'
  3 = 'LocalMarks1D'
   = ''
END_TEXTLIST

// ---- POUs/Print/DefGrid/_VISU_Templates/_VISU_ContainerDefGrid.TcVIS
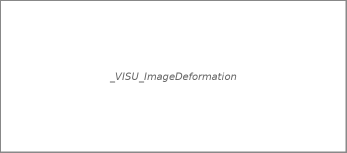
VISUALIZATION _VISU_ContainerDefGrid  // 347x153
VAR_IN_OUT
	m_Inst : FB_ContainerDefGrid;
END_VAR
    Frame (0,0 347x153)
        shows _VISU_ImageDeformation(m_Inst := m_Inst.fBImageDeformation)
END_VISUALIZATION

// ---- POUs/Print/DefGrid/_VISU_Templates/_VISU_CTsFlow.TcVIS
